// TIA Portal V17 program export: 1 tag tables, 0 data types, 0 data blocks, 10 code blocks (in call order from the OBs), 1 instance data blocks

VAR_GLOBAL   // PLC tag table "Default tag table"
END_VAR

ORGANIZATION_BLOCK "Main"   // OB1, LAD, ProgramCycle
TITLE = "Main Program Sweep (Cycle)"
{ S7_Optimized_Access := 'TRUE' }
VERSION : 0.1
// stored: AutoNumber true, IsIECCheckEnabled false, SetENOAutomatically false
   VAR_INPUT
      Initial_Call : Bool;   // Initial call of this OB
      Remanence : Bool;   // =True, if remanent data are available
   END_VAR
   VAR_TEMP
      SOME_BOOLEAN : Bool;
   END_VAR
BEGIN

REGION Network 1
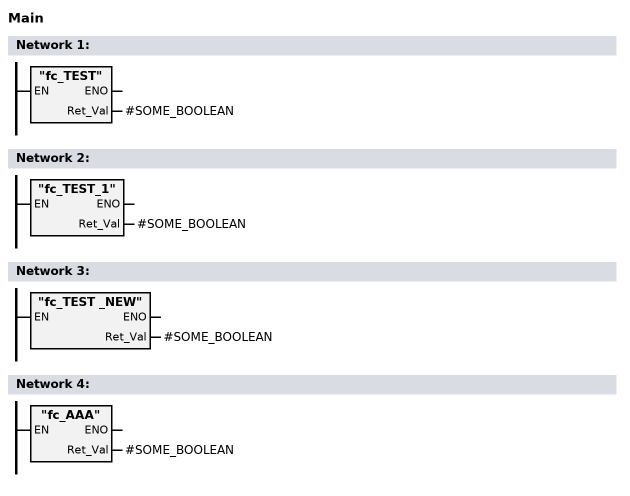
   RUNG wire#powerrail
      "fc_TEST"(Ret_Val => #SOME_BOOLEAN)
   END_RUNG
   // the same network as SCL:
   #SOME_BOOLEAN := "fc_TEST"();
END_REGION

REGION Network 2
   RUNG wire#powerrail
      "fc_TEST_1"(Ret_Val => #SOME_BOOLEAN)
   END_RUNG
   // the same network as SCL:
   #SOME_BOOLEAN := "fc_TEST_1"();
END_REGION

REGION Network 3
   RUNG wire#powerrail
      "fc_TEST _NEW"(Ret_Val => #SOME_BOOLEAN)
   END_RUNG
   // the same network as SCL:
   #SOME_BOOLEAN := "fc_TEST _NEW"();
END_REGION

REGION Network 4
   RUNG wire#powerrail
      "fc_AAA"(Ret_Val => #SOME_BOOLEAN)
   END_RUNG
   // the same network as SCL:
   #SOME_BOOLEAN := "fc_AAA"();
END_REGION
END_ORGANIZATION_BLOCK

FUNCTION "fc_TEST" : Bool

{ S7_Optimized_Access := 'TRUE' }
VERSION : 0.1
VAR_INPUT

END_VAR

VAR_OUTPUT

END_VAR

VAR_IN_OUT

END_VAR

VAR_TEMP

END_VAR

VAR CONSTANT

END_VAR


BEGIN
	REGION INITIAL_FUNCTION
	    #fc_TEST :=  NOT  TRUE;
	END_REGION
	
END_FUNCTION

FUNCTION "fc_TEST_1" : Bool

{ S7_Optimized_Access := 'TRUE' }
VERSION : 0.1
VAR_INPUT

END_VAR

VAR_OUTPUT

END_VAR

VAR_IN_OUT

END_VAR

VAR_TEMP

END_VAR

VAR CONSTANT

END_VAR


BEGIN
	REGION INITIAL_FUNCTION
	    #fc_TEST_1 := TRUE;
	END_REGION
	
END_FUNCTION

FUNCTION "fc_TEST _NEW" : Bool   // FC6, SCL
{ S7_Optimized_Access := 'TRUE' }
VERSION : 0.1
// stored: AutoNumber true, IsIECCheckEnabled false, SetENOAutomatically false, UDAEnableTagReadback false
BEGIN
   REGION RETURN_BOOLEAN
       #"fc_TEST _NEW" := FALSE;
   END_REGION
END_FUNCTION

FUNCTION "fc_AAA" : Bool   // FC7, SCL
{ S7_Optimized_Access := 'TRUE' }
VERSION : 0.1
// stored: AutoNumber true, IsIECCheckEnabled false, SetENOAutomatically false, UDAEnableTagReadback false
BEGIN
   #fc_AAA := true;
END_FUNCTION

FUNCTION "Block_1" : Void   // FC3, LAD
{ S7_Optimized_Access := 'TRUE' }
VERSION : 0.1
// stored: AutoNumber true, IsIECCheckEnabled false, SetENOAutomatically false, UDAEnableTagReadback false
   VAR_TEMP
      "A" : Bool;
      "B" : Bool;
   END_VAR
   VAR_TEMP   // added for the SCL form of the ladder/FBD networks
      _w1 : Bool;
   END_VAR
BEGIN

REGION Network 1
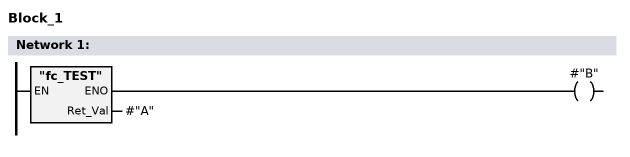
   RUNG wire#powerrail
      "fc_TEST"(Ret_Val => #"A")
      Coil( #"B" )
   END_RUNG
   // the same network as SCL:
   #"A" := "fc_TEST"(ENO => #_w1);
   #"B" := #_w1;
END_REGION
END_FUNCTION

FUNCTION "fc_CCC" : Void   // FC8, SCL
{ S7_Optimized_Access := 'TRUE' }
VERSION : 0.1
// stored: AutoNumber true, IsIECCheckEnabled false, SetENOAutomatically false, UDAEnableTagReadback false
BEGIN
END_FUNCTION

FUNCTION_BLOCK "Main_Safety_RTG1"   // FB1, F_FBD
{ S7_Optimized_Access := 'TRUE' }
VERSION : 0.1
// stored: AutoNumber false, IsIECCheckEnabled false, UDAEnableTagReadback false
BEGIN
END_FUNCTION_BLOCK

FUNCTION "fc_TEST_3" : Bool

{ S7_Optimized_Access := 'TRUE' }
VERSION : 0.1
VAR_INPUT

END_VAR

VAR_OUTPUT

END_VAR

VAR_IN_OUT

END_VAR

VAR_TEMP

END_VAR

VAR CONSTANT

END_VAR


BEGIN
	REGION INITIAL_FUNCTION
	    #fc_TEST_3 := TRUE;
	END_REGION
	
END_FUNCTION

FUNCTION "fc_TEST_2" : Bool

{ S7_Optimized_Access := 'TRUE' }
VERSION : 0.1
VAR_INPUT

END_VAR

VAR_OUTPUT

END_VAR

VAR_IN_OUT

END_VAR

VAR_TEMP

END_VAR

VAR CONSTANT

END_VAR


BEGIN
	REGION INITIAL_FUNCTION
	    #fc_TEST_2 := TRUE;
	END_REGION
	
END_FUNCTION

DATA_BLOCK "Main_Safety_RTG1_DB"   // DB1, F_DB
NAME : FUSI
VERSION : 0.1
// stored: AutoNumber true, DBAccessibleFromOPCUA true, DBAccessibleFromWebserver true, InstanceOfName Main_Safety_RTG1, InstanceOfType FB
"Main_Safety_RTG1"
BEGIN
END_DATA_BLOCK
